// TIA Portal V17 export
// export: Created 2025-06-26T06:33:57.9730409Z, ExportSetting WithDefaults, DisplayName Totally Integrated Automation Portal, DisplayVersion V17 Update 8, DisplayName TIA Portal Openness, DisplayVersion V17 Update 8, DisplayName TIA Portal Version Control Interface, DisplayVersion V17, DisplayName STEP 7 Professional, DisplayVersion V17 Update 8, DisplayName STEP 7 Safety, DisplayVersion V17 Update 6, DisplayName WinCC Advanced, DisplayVersion V17 Update 8
DATA_BLOCK "DB_ToHB"   // DB101
{ S7_Optimized_Access := 'FALSE' }
VERSION : 0.1
// stored: AutoNumber false, DBAccessibleFromOPCUA true, IsOnlyStoredInLoadMemory false, IsWriteProtectedInAS false
   VAR
      StartRequest : Bool;   // 1 = start Heatbooster, 0 = do nothing (level)
      StopRequest : Bool;   // 1 = stop, 0 = do nothing (overrides start signal) (level) (Regular stop, with cooldown periods etc)
      FastStopRequest : Bool;   // 1 = fast stop, 0 = do nothing (overrides start and stop signals) (level) (Stop NOW, but not Emergency Stop)
      EnableHeatbooster : Bool;   // 1 = allow operation, 0 = disable operation (level)
      AlarmAcknowledge : Bool;   // 1 = clear all alarms, 0 = do nothing (edge)
      ResetEmergencyStop : Bool;   // 1 = reset emergency stop, 0 = do nothing (edge)
      SpareCmd006 : Bool;   // 1 = Ventilation ok, 0 = ignore start command
      SpareCmd007 : Bool;   // 1 = Detected (stop request), 0 = do nothing
      SpareCmd010 : Bool;
      SpareCmd011 : Bool;
      SpareCmd012 : Bool;
      SpareCmd013 : Bool;
      SpareCmd014 : Bool;
      SpareCmd015 : Bool;
      SpareCmd016 : Bool;
      SpareCmd017 : Bool;
      WatchdogCounter : UInt;   // Liveness counter (free-running)
      Setpoint : Real;   // [%] Heatbooster setpoint
      SpareStatus080 : Bool;
      SpareStatus081 : Bool;
      SpareStatus082 : Bool;
      SpareStatus083 : Bool;
      SpareStatus084 : Bool;
      SpareStatus085 : Bool;
      SpareStatus086 : Bool;
      SpareStatus087 : Bool;
      SpareStatus090 : Bool;
      SpareStatus091 : Bool;
      SpareStatus092 : Bool;
      SpareStatus093 : Bool;
      SpareStatus094 : Bool;
      SpareStatus095 : Bool;
      SpareStatus096 : Bool;
      SpareStatus097 : Bool;
      Spare10 : Real;
      Spare14 : Real;
      Spare18 : Real;
      Spare22 : Real;
      Spare26 : Real;
      Spare30 : Real;
      Spare34 : Real;
      Spare38 : Real;
      ProteinDryerTemperature : Real;
      StarchDryerTemperature : Real;
      HBhallRelativeHumidity : Real;
      HBhallGasDetector : Real;
      StarchDryerAirInTemperature : Real;
      StarchDryerAirOutTemperature : Real;
      ProteinDryerAirInTemperature : Real;
      ProteinDryerAirOutTemperature : Real;
   END_VAR
BEGIN
END_DATA_BLOCK
